Fanuc TP program (LS listing): MAKRO050.LS

/PROG  MAKRO050
/ATTR
OWNER		= AUROM;
COMMENT		= "Inic. Marcas";
PROG_SIZE	= 3492;
CREATE		= DATE 00-03-13  TIME 16:56:34;
MODIFIED	= DATE 23-09-03  TIME 08:44:40;
FILE_NAME	= ;
VERSION		= 0;
LINE_COUNT	= 122;
MEMORY_SIZE	= 3784;
PROTECT		= READ_WRITE;
TCD:  STACK_SIZE	= 0,
      TASK_PRIORITY	= 50,
      TIME_SLICE	= 0,
      BUSY_LAMP_OFF	= 0,
      ABORT_REQUEST	= 0,
      PAUSE_REQUEST	= 0;
DEFAULT_GROUP	= *,*,*,*,*;
CONTROL_CODE	= 00000000 00000000;
/MN
   1:  !Inicializacion de Marcas ;
   2:  !Robot con Garra ;
   3:  !Soldadura Inductiva Est. ;
   4:  ! ;
   5:  !Control de Piezas ;
   6:  M[1]=((DI[603] AND DI[604] AND DI[605] AND DI[606]) OR DI[15]) ;
   7:  M[2]=(!DI[603] AND !DI[604] AND !DI[605] AND !DI[606]) ;
   8:  M[3]=((!DI[603] AND DI[604] AND DI[605] AND !DI[606]) OR DI[15]) ;
   9:  M[5]=((DI[603] AND !DI[604] AND !DI[605] AND DI[606]) OR DI[15]) ;
  10:  ! ;
  11:  !Control de Grupos de Sujecion ;
  12:  M[31]=(DI[579] AND !DI[580] AND DI[581] AND !DI[582] AND DI[583] AND !DI[584]) ;
  13:  M[32]=(!DI[579] AND DI[580] AND !DI[581] AND DI[582] AND !DI[583] AND DI[584]) ;
  14:  M[33]=(OFF) ;
  15:  M[34]=(OFF) ;
  16:  M[35]=(DI[585] AND !DI[586]) ;
  17:  M[36]=(!DI[585] AND DI[586]) ;
  18:  M[37]=(!DI[587] AND DI[588]) ;
  19:  M[38]=(DI[587] AND !DI[588]) ;
  20:  M[39]=(DI[589] AND !DI[590] AND DI[591] AND !DI[592]) ;
  21:  M[40]=(!DI[589] AND DI[590] AND !DI[591] AND DI[592]) ;
  22:  M[41]=(!DI[593] AND DI[594]) ;
  23:  M[42]=(DI[593] AND !DI[594]) ;
  24:  M[43]=(DI[595] AND !DI[596]) ;
  25:  M[44]=(!DI[595] AND DI[596]) ;
  26:  M[45]=(OFF) ;
  27:  M[46]=(OFF) ;
  28:  M[47]=(OFF) ;
  29:  M[48]=(OFF) ;
  30:  M[49]=(OFF) ;
  31:  M[50]=(OFF) ;
  32:  M[51]=(OFF) ;
  33:  M[52]=(OFF) ;
  34:  M[53]=(OFF) ;
  35:  M[54]=(OFF) ;
  36:  M[55]=(OFF) ;
  37:  M[56]=(OFF) ;
  38:  M[57]=(OFF) ;
  39:  M[58]=(OFF) ;
  40:  M[59]=(OFF) ;
  41:  M[60]=(OFF) ;
  42:  M[61]=(OFF) ;
  43:  M[62]=(OFF) ;
  44:  M[63]=((!DI[617] AND !DI[618]) OR DI[15]) ;
  45:  M[64]=(OFF) ;
  46:  M[65]=(OFF) ;
  47:  M[66]=(OFF) ;
  48:  M[67]=(OFF) ;
  49:  M[68]=(OFF) ;
  50:  ! ;
  51:  !Marcas de Usuario: ;
  52:  !Marca 1 ST1150 Vacia ;
  53:  M[10]=(!DI[60] AND DI[59] AND !DI[58] AND DI[57]) ;
  54:  !Marca 2 ST1150 C/Pieza 1 ;
  55:  M[11]=(DI[60] AND !DI[59] AND !DI[58] AND DI[57]) ;
  56:  !Marca 3 ST1150 Llena ;
  57:  M[12]=(DI[60] AND !DI[59] AND DI[58] AND !DI[57]) ;
  58:  !Marca 4 Estado de Garra ;
  59:  !Valvulas 1-7 en R ;
  60:  M[20]=(M[31] AND M[35] AND M[37] AND M[39] AND M[41] AND M[43]) ;
  61:  !Marca 5 Estado de Garra ;
  62:  !Valvula 1 en V, 2-7 en R ;
  63:  M[21]=(M[32] AND M[35] AND M[37] AND M[39] AND M[41] AND M[43]) ;
  64:  !Marca 6 Estado de Garra ;
  65:  !Valvula 1,2&5 en V, 3,4,6&7 en R ;
  66:  M[22]=(M[32] AND M[35] AND M[37] AND M[40] AND M[41] AND M[43] AND M[63]) ;
  67:  !Marca 7 Estado de Garra ;
  68:  !Valvula 1,2,3&5 en V, 4,6&7 en R ;
  69:  M[23]=(M[32] AND M[36] AND M[37] AND M[40] AND M[41] AND M[43] AND M[63]) ;
  70:  !Marca 8 Estado de Garra ;
  71:  !Valvula 1,2,3,5&6 en V, 4&7 en R ;
  72:  M[24]=(M[32] AND M[36] AND M[37] AND M[40] AND M[42] AND M[43] AND M[63]) ;
  73:  !Marca 9 Estado de Garra ;
  74:  !Valvula 2,3,5&6 en V, 1,4&7 en R ;
  75:  M[25]=(M[31] AND M[36] AND M[37] AND M[40] AND M[42] AND M[43] AND M[63]) ;
  76:  !Marca 10 Estado de Garra ;
  77:  !Valvula 4&6 en V, 1,2,3,5&7 en R ;
  78:  M[26]=(M[31] AND M[35] AND M[38] AND M[39] AND M[42] AND M[43]) ;
  79:  !Marca 11 Estado de Garra ;
  80:  !Valvulas 1-7 en R ;
  81:  M[27]=(M[32] AND M[35] AND !M[37] AND M[39] AND M[41] AND M[43]) ;
  82:  ! ;
  83:  M[28]=(M[32] AND M[35] AND M[37] AND M[40] AND M[41] AND M[43]) ;
  84:  ! ;
  85:   ;
  86:   ;
  87:   ;
  88:  !Seguridad de Maquina ;
  89:  M[30]=(DI[14] AND DI[24] AND DI[516]) ;
  90:  ! ;
  91:  !Soldadura Por Induccion ;
  92:  !Seguridad EZ1/SP1 ;
  93:  M[95]=(DI[705] AND !DI[706] AND DI[713] AND DI[714] AND ((!DI[715] AND DI[719]) OR DO[715]) AND !DI[773] AND !DI[779] AND DO[716]) ;
  94:  !Basculante 1 en Pos. de Reposo ;
  95:  M[96]=(DI[842] AND !DI[844] AND !DI[843] AND DI[845] AND !DO[715] AND (F[321] OR (DO[875] AND F[148]) OR (DO[1035] AND F[184]))) ;
  96:  !Flankenausw.der Fraeserumd.KF1 ;
  97:  M[97]=((DI[718] AND DO[718] OR F[312]) AND DI[834] AND DO[834] AND !F[72] AND !F[73] AND (F[90] OR F[92])) ;
  98:  ! ;
  99:  !EZ1/SP1/SZ1 Umdrehungen Startfr ;
 100:  R[2]=4    ;
 101:  !Umdrehungen Startfraesen Teil 2 ;
 102:  R[3]=4    ;
 103:  !Umdrehungen Nomalfraesen ;
 104:  R[4]=3    ;
 105:  !min. Oeffnung stat. EZ/SP ;
 106:  !beim Fraesen ;
 107:  R[60]=600    ;
 108:  ! ;
 109:  !;Ausgleichswert EZ1/SP1 ;
 110:  R[197]=106    ;
 111:  !Kappenverschl. Verhaeltnis ;
 112:  !feste EK in % (Stat-EZ1) ;
 113:  R[411]=65    ;
 114:   ;
 115:  !Kappenkompenstion bei ;
 116:  !stationaerer EZ1/SP1 ;
 117:  CALL MOTN004    ;
 118:  ! ;
 119:  !Aufruf Makro57 ;
 120:  CALL MAKRO057    ;
 121:  !Docking ;
 122:  CALL MAKRO058    ;
/POS
/END
